// TIA Portal V19 export
TYPE "UDT_STATUS_DIN"
   STRUCT
      switch : Bool;
      justActivated : Bool;
      justDectivated : Bool;
      fault : Bool;
      justHadFault : Bool;
      justLostFault : Bool;
      enabled : Bool;
      old : Struct
         switch : Bool;
         fault : Bool;
      END_STRUCT;
   END_STRUCT;
END_TYPE
